PROGRAM INTERNAL PRG_TESTS

(* Instantiate test suites here. Naming convention for tests should be a suffix with _Tests.
Good practice for creating test methods is to end them with _test as well. *)
VAR
	PathGeneratorTests		: FB_PathGenerator_Tests;
	UtilitiesTests			: FB_Utilities_Tests;
	FileHandlerTests		: FB_FileHandler_Tests;
	PathUtilitiesTests		: FB_PathUtilities_Tests;
	FileUtilitiesTests		: FB_FileUtilities_Tests;
	DirectoryUtilitiesTests	: FB_DirectoryUtilities_Tests;
END_VAR

VAR CONSTANT
	FILE_HANDLER_TESTS_PATH			: Tc2_System.T_MaxString := '/home/Administrator/ZigaLibsTestFolder/FileHandlerTests/';
	FILE_HANDLER_TESTS_DIRECTORY	: Tc2_System.T_MaxString := '/home/Administrator/ZigaLibsTestFolder/FileHandlerTests';
	NET_ID							: Tc2_System.T_AmsNetID := '';
	DATE_TIME_MAX_VALUE				: DT  := DATE_AND_TIME#2106-02-07-06:28:15;
END_VAR

// Run tests in parallel
//TcUnit.RUN();

// Run tests in sequence, one after the other.
TcUnit.RUN_IN_SEQUENCE();

END_PROGRAM

(* stored: Version 1.1.0.1, ProductVersion 3.1.4024.15
   POU PRG_TESTS: Id {fa45e8d0-6cda-46ca-bddb-e3c59f6853b2}, SpecialFunc None *)
